// TIA Portal V19 export
DATA_BLOCK "HmiInterface"   // DB47
// stored: MemoryReserve 100, Namespace Unit.Em1
   VAR
      em : "LAF_typeEmInterface";
      jobs : "LAF_typeJobsInterface";
      sequence : "LAF_typeSequenceInterface";
   END_VAR
BEGIN
END_DATA_BLOCK
